// TIA Portal V16 export
// export: Created 2021-10-10T10:54:05.2283245Z, ExportSetting None, DisplayName Totally Integrated Automation Portal, DisplayVersion V16, DisplayName TIA Portal Version Control Interface, DisplayVersion V16, DisplayName TIA Portal Openness, DisplayVersion V16, DisplayName STEP 7 Professional, DisplayVersion V16, DisplayName STEP 7 Safety, DisplayVersion V16, DisplayName WinCC Advanced, DisplayVersion V16
FUNCTION "fcTest" : Void   // FC1, LAD
{ S7_Optimized_Access := 'TRUE' }
// stored: SetENOAutomatically false
   VAR_TEMP
      tBool : Bool;
   END_VAR
   VAR CONSTANT
      CONSTANT_BOOL : Bool := TRUE;
   END_VAR
BEGIN

REGION Network 1
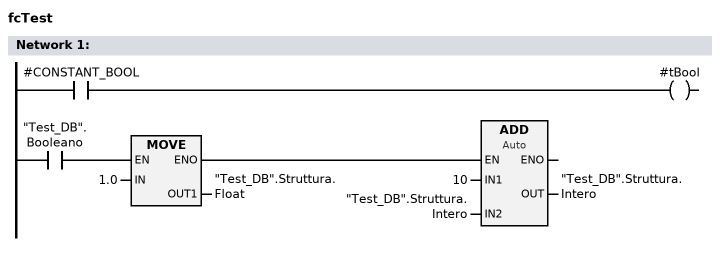
   RUNG wire#powerrail
      Contact( #CONSTANT_BOOL )
      Coil( #tBool )
   END_RUNG
   RUNG wire#powerrail
      Contact( "Test_DB".Booleano )
      Move(in := 1.0, out1 => "Test_DB".Struttura.Float)
      Add(in1 := 10, in2 := "Test_DB".Struttura.Intero, out => "Test_DB".Struttura.Intero)
   END_RUNG
   // the same network as SCL:
   #tBool := #CONSTANT_BOOL;
   IF "Test_DB".Booleano THEN
       "Test_DB".Struttura.Float := 1.0;
       "Test_DB".Struttura.Intero := 10 + "Test_DB".Struttura.Intero;
   END_IF;
END_REGION
END_FUNCTION
